// TwinCAT 3 PLC project BE_TheresianumPLCCode
// ProgramVersion: 3.1.4024.0
// libraries:
//   EfficientIO Communicator, * (EfficientIO)
//   EfficientIO Energy Basic, * (EfficientIO)
//   EfficientIO ModbusTCP, * (EfficientIO)
//   Lynus Persistent Data V1, * (Lynus AG)
//   Lynus Standards, * (EfficientIO)
//   Tc2_Standard, * (Beckhoff Automation GmbH)
//   Tc2_System, * (Beckhoff Automation GmbH)
//   Tc3_Module, * (Beckhoff Automation GmbH)
// project tree:
//   / FastTask.TcTTO, MiddleTask.TcTTO, SlowTask.TcTTO
//   POUs/ MAIN.TcPOU, prgComEffIO.TcPOU, prgEM.TcPOU, prgRWEffIO.TcPOU, prgVarEffIO.TcPOU
// real-time tasks:
//   TASK FastTask: cycle T#5ms, priority 6, ADS port 350
//   TASK MiddleTask: cycle T#10ms, priority 8, ADS port 351
//   TASK SlowTask: cycle T#20ms, priority 10, ADS port 352

CONFIGURATION BE_TheresianumPLCCode
    RESOURCE PLC ON TwinCAT3
        TASK FastTask(INTERVAL := T#5ms, PRIORITY := 6);
        TASK MiddleTask(INTERVAL := T#10ms, PRIORITY := 8);
        TASK SlowTask(INTERVAL := T#20ms, PRIORITY := 10);
        PROGRAM prgVarEffIO WITH FastTask : prgVarEffIO;
        PROGRAM prgRWEffIO WITH FastTask : prgRWEffIO;
        PROGRAM prgComEffIO WITH SlowTask : prgComEffIO;
    END_RESOURCE
END_CONFIGURATION

// ---- POUs/prgVarEffIO.TcPOU
PROGRAM prgVarEffIO
VAR
	fbVar		: FB_VarInfo_V3;
END_VAR

fbVar(
	bReadInfo:= , 
	eTMCFile:= eSelectTMCFile.eDontUseTMCFile, 
	eSavePositionTMCFile:= eSavePositionOnPLC.ePostionHardDisk, 
	udiCounterFoundVariables=> , 
	bError=> , 
	bBusy=> , 
	byProgress=> , 
	udiErrorCodeOut=> , 
	eErrorVarInfo_Out=> , 
	sVarWithError=> );

END_PROGRAM

// ---- POUs/prgRWEffIO.TcPOU
PROGRAM prgRWEffIO
VAR
	fbRW1		: FB_ReadWrite_V2;
END_VAR

fbRW1(
	eUploadType:= eSelectDataUploadType.e_Change_Intervall5min, 
	bBusy=> , 
	bError=> , 
	udiErrorCodeOut=> , 
	eErrorReadWrite_Out=> );

END_PROGRAM

// ---- POUs/prgComEffIO.TcPOU
PROGRAM prgComEffIO
VAR
	fbCom		: FB_MqttCommunicator_V3;
END_VAR

fbCom(
	bConnect:= TRUE, 
	strAuthKey:=  'EIO08031879806' , 
	sUserName:= 'bd8cddef-7a46-4cb7-9100-c3c67f8ed94a', 
	sUserPassword:= '26bcb4df-2135-49e0-bf55-9c706b8073f9', 
	eSavePositionCertificate:= eSavePositionOnPLC.ePostionC, 
	time_HeartBeat_sec := T#1S,
	bConnected=> , 
	bError=> , 
	hrErrorCode=> , 
	eConnectionState=> , 
	eErrorMessage_Out=> );

END_PROGRAM

// ---- POUs/MAIN.TcPOU
PROGRAM MAIN
VAR
END_VAR

END_PROGRAM

// ---- POUs/prgEM.TcPOU
PROGRAM prgEM
VAR
	FB_Phoenix:FB_PhoenixContact_EM_EEM_EM375;
	
	
	
	lrPower_Grid_TotalkW		: LREAL;			//{#lynus.ag#()}
	lrPower_Grid_L1				: LREAL;			//{#lynus.ag#()}
	lrPower_Grid_L2				: LREAL;			//{#lynus.ag#()}
	lrPower_Grid_L3				: LREAL;			//{#lynus.ag#()}
	lrCurrent_Grid_L1			: LREAL;			//{#lynus.ag#()}
	lrCurrent_Grid_L2			: LREAL;			//{#lynus.ag#()}
	lrCurrent_Grid_L3			: LREAL;			//{#lynus.ag#()}
	lrVoltage_Grid_L1N			: LREAL;			//{#lynus.ag#()}
	lrVoltage_Grid_L2N			: LREAL;			//{#lynus.ag#()}
	lrVoltage_Grid_L3N			: LREAL;			//{#lynus.ag#()}
	

	flEMPowerTotal				: LREAL;
	bPullSuccessfull 			: BOOL;
	udintErrorID				: UDINT;


	uint_State			AT%I* 	: UINT;
	lrPower_House_kW			: LREAL;			//{#lynus.ag#()}
		
END_VAR

VAR PERSISTENT
	bEnableEM			: 	BOOL;
END_VAR


// lrPower_House_kW := LIMIT(0,lrPower_Grid_TotalkW - prgCS1.lrPower_Alfen_1_S1 + prgPV.lrPower_PV_kW,100);


FB_Phoenix(
	bEnable:= TRUE, 
	byUnitID:= 255, 
	sIPAdress:= '192.168.1.11', 
	stDataEMPower=> , 
	stDataEMCounter=> , 
	stDataEMPowerRealTime=> , 
	stDataEMCounterRealTime=> , 
	diNrOfEM_OUT=> );

lrPower_Grid_TotalkW 	:= 	FB_Phoenix.stDataEMPower.lrPowerTotal;
lrPower_Grid_L1		 	:= 	FB_Phoenix.stDataEMPower.lrPowerL1;
lrPower_Grid_L2		 	:= 	FB_Phoenix.stDataEMPower.lrPowerL2;
lrPower_Grid_L3		 	:= 	FB_Phoenix.stDataEMPower.lrPowerL3;
lrCurrent_Grid_L1 		:= 	FB_Phoenix.stDataEMPower.lrCurrentL1;
lrCurrent_Grid_L2 		:= 	FB_Phoenix.stDataEMPower.lrCurrentL2;
lrCurrent_Grid_L3 		:= 	FB_Phoenix.stDataEMPower.lrCurrentL3;
lrVoltage_Grid_L1N		:= 	FB_Phoenix.stDataEMPower.lrVoltageL1N;
lrVoltage_Grid_L2N		:= 	FB_Phoenix.stDataEMPower.lrVoltageL2N;
lrVoltage_Grid_L3N		:= 	FB_Phoenix.stDataEMPower.lrVoltageL3N;

END_PROGRAM
